FUNCTION_BLOCK FB_AnnealingOven
VAR_INPUT
END_VAR
VAR_OUTPUT
END_VAR
VAR
END_VAR

END_FUNCTION_BLOCK

(* stored: Version 1.1.0.1, ProductVersion 3.1.4024.10
   POU FB_AnnealingOven: Id {55cd34b0-1d7f-435c-9435-b7ad14b8fb75}, SpecialFunc None *)
